FUNCTION_BLOCK FB_Motor

VAR_STAT
	nNum : INT;
END_VAR
VAR
	{attribute 'hide'}
	bStart : BOOL := TRUE;
END_VAR

METHOD Start : BOOL
VAR_INPUT
END_VAR
nNum := nNum + 1;
END_METHOD

END_FUNCTION_BLOCK

(* stored: Version 1.1.0.1, ProductVersion 3.1.4024.16
   POU FB_Motor: Id {a23ca182-15e8-4e99-91c3-848ac3b0a8af}, SpecialFunc None
   Method Start: Id {69721c44-875e-461f-8521-a56654156274} *)
